(* IEC 61131-3 sources: tgTCLogLib/, 3 files *)

(* ---- ST_funcs.BSD.iecst ---- *)
{attribute 'dllimport', 'tgLogLib.so'}
FUNCTION tgLog_MQTT_Init : DINT
    VAR_INPUT
        broker : STRING(255);
        port : DINT;
        clientID : STRING(255);
    END_VAR
END_FUNCTION

{attribute 'dllimport', 'tgLogLib.so'}
FUNCTION tgLog_MQTT_Log : DINT
    VAR_INPUT
        topic : STRING(255);
        message : STRING(255);
    END_VAR
END_FUNCTION

{attribute 'dllimport', 'tgLogLib.so'}
FUNCTION tgLog_MQTT_Close : VOID
END_FUNCTION

{attribute 'dllimport', 'tgLogLib.so'}
FUNCTION tgLog_REST_Post : DINT
    VAR_INPUT
        url : STRING(255);
        jsonPayload : STRING(1024);
    END_VAR
END_FUNCTION

{attribute 'dllimport', 'tgLogLib.so'}
FUNCTION tgLog_MySQL_Connect : DINT
    VAR_INPUT
        host : STRING(255);
        user : STRING(255);
        password : STRING(255);
        database : STRING(255);
    END_VAR
END_FUNCTION

{attribute 'dllimport', 'tgLogLib.so'}
FUNCTION tgLog_MySQL_Log : DINT
    VAR_INPUT
        table : STRING(255);
        columns : STRING(255);
        values : STRING(255);
    END_VAR
END_FUNCTION

{attribute 'dllimport', 'tgLogLib.so'}
FUNCTION tgLog_MySQL_Close : VOID
END_FUNCTION

{attribute 'dllimport', 'tgLogLib.so'}
FUNCTION tgLog_InfluxDB_Write : DINT
    VAR_INPUT
        host : STRING(255);
        port : DINT;
        database : STRING(255);
        measurement : STRING(255);
        fields : STRING(1024);
        tags : STRING(255);
    END_VAR
END_FUNCTION

(* ---- ST_funcs.Windows.iecst ---- *)
{attribute 'dllimport', 'tgLogLib.dll'}
FUNCTION tgLog_MQTT_Init : DINT
    VAR_INPUT
        broker : STRING(255);
        port : DINT;
        clientID : STRING(255);
    END_VAR
END_FUNCTION

{attribute 'dllimport', 'tgLogLib.dll'}
FUNCTION tgLog_MQTT_Log : DINT
    VAR_INPUT
        topic : STRING(255);
        message : STRING(255);
    END_VAR
END_FUNCTION

{attribute 'dllimport', 'tgLogLib.dll'}
FUNCTION tgLog_MQTT_Close : VOID
END_FUNCTION

{attribute 'dllimport', 'tgLogLib.dll'}
FUNCTION tgLog_REST_Post : DINT
    VAR_INPUT
        url : STRING(255);
        jsonPayload : STRING(1024);
    END_VAR
END_FUNCTION

{attribute 'dllimport', 'tgLogLib.dll'}
FUNCTION tgLog_MySQL_Connect : DINT
    VAR_INPUT
        host : STRING(255);
        user : STRING(255);
        password : STRING(255);
        database : STRING(255);
    END_VAR
END_FUNCTION

{attribute 'dllimport', 'tgLogLib.dll'}
FUNCTION tgLog_MySQL_Log : DINT
    VAR_INPUT
        table : STRING(255);
        columns : STRING(255);
        values : STRING(255);
    END_VAR
END_FUNCTION

{attribute 'dllimport', 'tgLogLib.dll'}
FUNCTION tgLog_MySQL_Close : VOID
END_FUNCTION

{attribute 'dllimport', 'tgLogLib.dll'}
FUNCTION tgLog_InfluxDB_Write : DINT
    VAR_INPUT
        host : STRING(255);
        port : DINT;
        database : STRING(255);
        measurement : STRING(255);
        fields : STRING(1024);
        tags : STRING(255);
    END_VAR
END_FUNCTION

(* ---- example.iecst ---- *)
PROGRAM MAIN
VAR
    result : DINT;
END_VAR

// MQTT-Logging
result := tgLog_MQTT_Init('broker.example.com', 1883, 'TwinCATClient');
result := tgLog_MQTT_Log('test/topic', 'Hello MQTT');
tgLog_MQTT_Close();

// REST API Logging
result := tgLog_REST_Post('http://example.com/api/log', '{"key": "value"}');

// InfluxDB Logging
result := tgLog_InfluxDB_Write('127.0.0.1', 8086, 'myDatabase', 'temperature', 'value=25.3', 'sensor=1');

// MySQL Logging
result := tgLog_MySQL_Connect('127.0.0.1', 'user', 'password', 'myDatabase');
result := tgLog_MySQL_Log('measurements', 'timestamp, value', '"2025-01-15 12:00:00", 42');
tgLog_MySQL_Close();
